{attribute 'qualified_only'}
{attribute 'strict'}
TYPE eStationState :
(
	Alarm 		:= -1,
	Disable 	:= 0,
	Ready 		:= 1,
	Working		:= 2,
	EndOfJob	:= 3,
	Undefine	:= 4,
	Extraction	:= 5,
	Infeed		:= 6
);
END_TYPE

(* stored: Version 1.1.0.1, ProductVersion 3.1.4024.13
   DUT eStationState: Id {502f3067-ec99-4d87-81d8-b0a7e1677ed2} *)
